// TwinCAT 3 PLC project PlcIotHttpSamplesAwsSigV4
// ProgramVersion: 3.1.4024.12
// libraries:
//   Tc2_Standard, * (Beckhoff Automation GmbH)
//   Tc2_System, * (Beckhoff Automation GmbH)
//   Tc3_IotBase, * (Beckhoff Automation GmbH)
//   Tc3_Module, * (Beckhoff Automation GmbH)
// project tree:
//   / PlcTask.TcTTO (not stored)
//   POUs/AWS Sig V4/ FB_TestHTTP_Get_AwsSigV4.TcPOU
//   POUs/ MAIN.TcPOU
// (motion and I/O tree: see PLC project plciothttpsamplespostman)
// real-time tasks:
//   TASK PlcTask: cycle T#10ms, priority 20, ADS port 350
//   TASK PlcTask1: cycle T#10ms, priority 21, ADS port 351
//   TASK PlcTask2: cycle T#10ms, priority 22, ADS port 352
//   TASK PlcTask3: cycle T#10ms, priority 23, ADS port 353
//   TASK PlcTask4: cycle T#10ms, priority 24, ADS port 354
//   TASK PlcTask5: cycle T#10ms, priority 25, ADS port 355
//   TASK PlcTask6: cycle T#10ms, priority 26, ADS port 356

// ---- POUs/AWS Sig V4/FB_TestHTTP_Get_AwsSigV4.TcPOU
FUNCTION_BLOCK FB_TestHTTP_Get_AwsSigV4
VAR_INPUT
	bSend				: BOOL;
END_VAR
VAR_IN_OUT
	fbClient			: FB_IotHttpClient;
END_VAR
VAR_OUTPUT
	bBusy				: BOOL;
	bError				: BOOL;
END_VAR
VAR
	fbRequest			: FB_IotHttpRequest;
	fbSig4Header		: FB_IotHttpAwsSig4HeaderFieldMap;
	nState				: UDINT;
	RisingEdge			: R_TRIG;
	
	bGetContentResult	: BOOL;
	sContent			: STRING(5000);
	
	bGetJsonResult		: BOOL;
	sResultValue		: STRING;
	
	nReqCount			: UDINT;	
	nResCount			: UDINT;
	nValidResCount		: UDINT;
	nErrCount			: UDINT;
	sRequestUrl			: STRING(500):='?Action=RunInstances&ImageId=ami-0229f7666f517b31e&InstanceType=t2.small&KeyName=Test&MaxCount=1&MinCount=1&Version=2016-11-15';
	//sRequestUrl			: STRING(500):='?Action=DescribeInstances&Version=2016-11-15';
	sService			: STRING:='ec2';
	sRegion				: STRING:='us-east-1';
	sAccessKey			: STRING:='censored';
	sSecretKey			: STRING:='censored';
	sSignedHeaders		: STRING:='host;x-amz-date';
	bSetParameter		: BOOL;
END_VAR

RisingEdge(CLK:= bSend );

CASE nState OF
0:	
	IF RisingEdge.Q THEN 
		bSetParameter:=fbSig4Header.SetParameter(sService, sRegion, sAccessKey, sSecretKey, sSignedHeaders);	
		IF bSetParameter THEN
			IF fbRequest.SendRequest(sUri:=sRequestUrl, fbClient:=fbClient, eRequestType:=ETcIotHttpRequestType.HTTP_Get, 0, 0, fbHeader:=fbSig4Header) THEN				
				nState:= 1;
				nReqCount:= nReqCount+1;
				bBusy:= TRUE;
				bError:= FALSE;
			END_IF
			bSetParameter:=FALSE;	
		END_IF
				
	END_IF
1:
	IF NOT fbRequest.bBusy THEN
		bError:= TRUE;
		IF NOT fbRequest.bError THEN				 
			bGetContentResult:= fbRequest.GetContent(pContent:= ADR(sContent), nContentSize:= SIZEOF(sContent), bSetNullTermination:= TRUE);
			IF fbRequest.nStatusCode >= 200 AND fbRequest.nStatusCode < 300 THEN				
				nResCount:= nResCount+1;
				// do something with XML response
				bError:=FALSE;			
			END_IF
		END_IF
		nState:= 0;
		bBusy:= FALSE;
		IF bError THEN
			nErrCount:= nErrCount+1;
		END_IF
	END_IF  	
END_CASE

END_FUNCTION_BLOCK

// ---- POUs/MAIN.TcPOU
PROGRAM MAIN
VAR
	// trigger command execution for AWS Sig V4 samples
	bGetAWSSigV4					: BOOL;

	fbHttpClientAWSSigV4			: FB_IotHttpClient :=(sHostName:='ec2.us-east-1.amazonaws.com',
									bKeepAlive:=FALSE, tConnectionTimeout:=T#10S);

	fbHttpGetAWSSigV4				: FB_TestHTTP_Get_AwsSigV4;
END_VAR

//init client parameters at startup
IF NOT fbHttpClientAWSSigV4.bConfigured THEN
	fbHttpClientAWSSigV4.nHostPort:=443;
	fbHttpClientAWSSigV4.stTLS.bNoServerCertCheck:=TRUE;
END_IF

IF fbHttpClientAWSSigV4.bConfigured THEN
	fbHttpGetAWSSigV4(bSend:=bGetAWSSigV4, fbClient:=fbHttpClientAWSSigV4);
END_IF

fbHttpClientAWSSigV4.Execute();

END_PROGRAM
